FUNCTION_BLOCK FB_Camera
VAR
	fbCamera : FB_VN_SimpleCameraControl;
	
	eState				:	Tc3_Vision.ETcVnCameraState;

//HResult
	{attribute 'displaymode':='hex'}
	hr					: 	HResult;
	{attribute 'displaymode':='hex'}
	hrWD_LocatePuck		:	HResult;
	{attribute 'displaymode':='hex'}
	hrLocatePuck		:	HResult;
	{attribute 'displaymode':='hex'}	
	hrDraw				: 	HResult;
	{attribute 'displaymode':='hex'}	
	hrCircle			:	HResult;
	{attribute 'displaymode':='hex'}
	hrWD_Threshold		:	HResult;
	{attribute 'displaymode':='hex'}	
	hrThreshold			:	HResult;
	{attribute 'displaymode':='hex'}	
	hrWD_Filter			:	HResult;	
	{attribute 'displaymode':='hex'}	
	hrFilter			:	HResult;
	{attribute 'displaymode':='hex'}	
	hrMorph				: 	HResult;
	{attribute 'displaymode':='hex'}
	hrWD_Contour		: 	HResult;
	{attribute 'displaymode':='hex'}	
	hrContour			: 	HResult;
	{attribute 'displaymode':='hex'}
	hrMatch				:	HResult;
		
// Colors	 
	aColorWhite			: 	TcVnVector4_LREAL := [255, 255, 255];
	aColorBlack			: 	TcVnVector4_LREAL := [0, 0, 0];
	aColorGreen			: 	TcVnVector4_LREAL := [0, 175, 0];
	aColorBlue			: 	TcVnVector4_LREAL := [0, 0, 255];
	aColorRed			: 	TcVnVector4_LREAL := [255, 0, 0];
	aColorMagenta		: 	TcVnVector4_LREAL := [255, 0, 255];
	
//images
	ipImageIn			:	ITcVnImage;
	ipImageWork			:	ITcVnImage;
	ipImageThreshold	:	ITcVnImage;	
	ipImageFilter		:	ITcVnImage;
	ipImageResult		:	ITcVnImage;
	
	ipImageInDisp		:	ITcVnDisplayableImage;
	ipImageWorkDisp		:	ITcVnDisplayableImage;
	ipImageThresDisp	:	ITcVnDisplayableImage;
	ipImageFilterDisp	:	ITcVnDisplayableImage;
	ipImageResultDisp	:	ITcVnDisplayableImage;
	
//Containers
	ipBlobContourPuckList: 	ITcVnContainer;
	ipInnercontourList	:	ITcVnContainer;	
	
//Contours
	ipPuckContour		: 	ITcVnContainer;
	ipInnerContour		:	ITcVnContainer;
	ipCompareContour	:	ITcVnContainer;
	
//iterators
	ipIterator			:	ITcVnForwardIterator;
	
//Blob parameters
	stBlobParamsPuck	: 	TcVnParamsBlobDetection;
	stBlobParamsInner	:	TcVnParamsBlobDetection;

//Watchdog variables
	tStop_LocatePuck	: 	DINT;
	nFraction_Locate	: 	UDINT;
	tRest_Locate		: 	DINT;

	tStop_Threshold		: 	DINT;
	nFraction_Threshold	: 	UDINT;
	tRest_Threshold		: 	DINT;

	tStop_filter		:	DINT;
	nFraction_Filter	:	UDINT;
	tRest_Filter		:	DINT;
	
	tStop_Contour		: 	DINT;
	nFraction_Contour	: 	UDINT;
	tRest_Contour		: 	DINT;

	
//Puck variables
	nNumOfElemPuck		: 	ULINT;
	PuckCenter			: 	TcVnPoint2_REAL;
	PuckRadius			: 	REAL;
	
//Threshold variables
	fThreshold			: 	LREAL;
	eThresholdType		: 	ETcVnThresholdType;
	
//Morph variables
	eOperator			: 	ETcVnMorphologicalOperator;
	ipElement			: 	ITcVnImage;
	eSEShape			: 	ETcVnStructuringElementShape;
	aSESize				: 	ARRAY [0..1] OF UDINT;

//Compare containers
	fbLoadContour		:	FB_VN_ReadContainer; //used to load the contour to compare to
	fDissimilarity		: 	LREAL;

//ROI settings
	bROI				: 	BOOL;
	aOffsetROI 			: 	TcVnPoint2_DINT;
	aOffsetROISize 		: 	TcVnPoint2_DINT := [460,460];
	aOffsetROIDraw 		: 	TcVnPoint2_DINT;

//Timetracking
	CPUTime 			: 	GETCPUCOUNTER;
	udStartTime			: 	UDINT;
	udEndTime			: 	UDINT;
	sTime				: 	STRING;
	
//Other Variables
	bFirstScan			: 	BOOL := TRUE;		
	bNewImageIn			: 	BOOL;				//check if there is a new image
	nImageCount			: 	LINT;
	fArea				: 	LREAL;
	aOffsetContour		: 	TcVnPoint;
	sPassString			: 	STRING;
	bMatch				: 	BOOL;
	nNumOfElemInner		: 	ULINT;

END_VAR

//LAB 3-1 START

IF bFirstScan THEN

// Blob Params for Puck Detection
	stBlobParamsPuck.bFilterByArea			:=  TRUE;
	stBlobParamsPuck.fMinArea       		:=  350_000;
	stBlobParamsPuck.fMaxArea       		:=  600_000;
	stBlobParamsPuck.bFilterByCircularity	:=  TRUE;
	stBlobParamsPuck.fMinCircularity		:=  0.8;
	stBlobParamsPuck.fMaxCircularity		:=  1;
	
//Blob Params for Inner Detection
	stBlobParamsInner.bFilterByArea	:=  TRUE;
	stBlobParamsInner.fMinArea       :=  30_000;
	stBlobParamsInner.fMaxArea       :=  120_000;


//watchdogSettings	
	tStop_LocatePuck 						:= 	5000;
	tStop_Threshold							:=	5000;
	tStop_Filter							:=	5000;
	tStop_Contour							:=	5000;

//Threshold setting
	fThreshold 								:= 	60;
	eThresholdType 							:=	TCVN_TT_BINARY;	

//Morph settings
	eOperator 								:= 	TCVN_MO_CLOSING;
	eSEShape 								:= 	TCVN_SES_RECTANGLE;	
	aSESize[0]								:=	8;
	aSESize[1]								:= 	8;
	
//Create element for Morph
	hr := F_VN_CreateStructuringElement(
		ipStructuringElement    :=  ipElement,
		eShape                  :=  eSEShape,
		nWidth					:=	aSESize[0],
		nHeight					:=	aSESize[1],
		hrPrev                  :=  hr);

	fbLoadContour(
		sFilePath:= 'C:\EngineeringWeek2023 Vision/Arm.xml', 
		ipDestContainer:= ipCompareContour, 
		nDestTypeGuid:= , 
		bRead:= TRUE, 
		nTimeout:= , 
		bBusy=> , 
		bError=> , 
		nErrorId=> );
		
	IF NOT fbLoadContour.bBusy AND NOT fbLoadContour.bError THEN
		fbLoadContour(sFilePath:= 'C:\TcVision_Contour_Files/Arm.xml', bRead := FALSE);	
		bFirstScan 								:= 	FALSE;
	END_IF
END_IF

//LAB 3-1 END

//LAB 2 START
bNewImageIn := FALSE;

eState := fbCamera.GetState();

CASE eState OF

	ETcVnCameraState.TCVN_CS_ERROR:
		hr := fbCamera.Reset();		


	ETcVnCameraState.TCVN_CS_INITIAL,
	ETcVnCameraState.TCVN_CS_INITIALIZING,
	ETcVnCameraState.TCVN_CS_INITIALIZED,
	ETcVnCameraState.TCVN_CS_OPENING, 
	ETcVnCameraState.TCVN_CS_OPENED, 
	ETcVnCameraState.TCVN_CS_STARTACQUISITION:
		hr := fbCamera.StartAcquisition();
	
	ETcVnCameraState.TCVN_CS_ACQUIRING,
	ETcVnCameraState.TCVN_CS_TRIGGERING:
		hr := fbCamera.GetCurrentImage(ipImageIn); // get image from buffer thats stored in ipImageIn
		IF SUCCEEDED(hr) AND ipImageIn <> 0 THEN
			nImageCount := nImageCount +1;
			bNewImageIn := TRUE;
		END_IF
		IF eState = 9 THEN		//triggering
			hr := fbCamera.TriggerImage();
			// After a Software Trigger, Camera enters Triggering Mode and acquires and sends an image
			// The Software Trigger must be called again to complete the transition back to Acquiring mode
			// This also applies to the File Source Control when in Trigger mode
		END_IF

END_CASE

IF bNewImageIn THEN
	
	CPUTime(cpuCntLoDW => udStarttime);
//Image Manipulation
	//Copy image into displayable image
	hr := F_VN_CopyIntoDisplayableImage(ipImageIn,ipImageInDisp,hr);


	//Copy image to new image to write results in
	hr := F_VN_CopyImage(ipImageIn, ipImageResult,hr);
//END_IF
//LAB 2 END

//LAB 3-2 START	
	//turn image into a grayscale image
	hr := F_VN_ConvertColorSpace(ipImageIn, ipImageWork, TCVN_CST_RGB_TO_GRAY, hr);
	hr := F_VN_CopyIntoDisplayableImage(ipImageWork,ipImageWorkDisp,hr);
	
	//find the whole puck
	hrWD_LocatePuck := F_VN_StartRelWatchdog(tStop_LocatePuck, hr);
		hrLocatePuck := F_VN_DetectBlobs(
			ipSrcImage		:= ipImageWork,
			ipBlobContours	:= ipBlobContourPuckList,
			stParams		:= stBlobParamsPuck,
			hrPrev			:= hr);
	hrWD_LocatePuck := F_VN_StopWatchdog(hrWD_LocatePuck, nFractionProcessed=>nFraction_Locate, tRest=>tRest_Locate);

	hr := F_VN_GetNumberOfElements(ipBlobContourPuckList, nNumOfElemPuck, S_OK);
	
	IF nNumOfElemPuck > 0 THEN
		
		
		
		
		//F_VN_GetAt.. (Get a single oontour out of a container)

		hr := F_VN_GetAt_ITcVnContainer(
			ipSrcContainer		:= ipBlobContourPuckList,
			ipDestContainer		:= ipPuckContour,
			nIndex				:= 0,		//first contour out of the container
			hrPrev				:= hr);
		

		//find enclosing circle (for center point and radius)
		hrCircle := F_VN_EnclosingCircle(
			ipPointSet	:= ipPuckContour,
			aCenter		:= PuckCenter,
			fRadius		:= PuckRadius,
			hrPrev		:= hr);
		
		//draw shape and center of puck
		hrDraw := F_VN_DrawContours(ipBlobContourPuckList, -1, ipImageResult, aColorRed, 3,hrCircle);
		hrDraw := F_VN_DrawPointExp(REAL_TO_UDINT(PuckCenter[0]), REAL_TO_UDINT(PuckCenter[1]), ipImageResult, 2, aColorMagenta, 40, 5, 8, hrDraw);
		hr := F_VN_CopyIntoDisplayableImage(ipImageResult,ipImageResultDisp,hrDraw);


		
	END_IF

//LAB 3-2 END

END_FUNCTION_BLOCK

(* stored: Version 1.1.0.1, ProductVersion 3.1.4024.12
   POU FB_Camera: Id {a541b016-bf05-4d4a-a2b6-a489256debc2}, SpecialFunc None *)
